FUNCTION F_WordSwap : DWORD
VAR_INPUT
	nDataIn : DWORD;
END_VAR
VAR
	nHighWord : WORD;
	nLowWord : WORD;
END_VAR

nLowWord := DWORD_TO_WORD(nDataIn);
nHighWord := DWORD_TO_WORD( SHR(nDataIn, 16 ));

F_WordSwap := nHighWord + nLowWord;

END_FUNCTION

(* stored: Version 1.1.0.1, ProductVersion 3.1.4022.3
   POU F_WordSwap: Id {75adb5c7-1721-4a35-afe6-e1568ba4a27e}, SpecialFunc None *)
